{attribute 'reflection'}
FUNCTION_BLOCK FBEvent
VAR_INPUT
END_VAR
VAR_OUTPUT
END_VAR
VAR
  runner: REFERENCE TO EventRunner;
  {attribute 'instance-path'}
  {attribute 'noinit'}
  path: STRING(255);
  id: INT;
  _message: STRING(255);
END_VAR

METHOD add_message
VAR_INPUT
  level: EventLevel;
END_VAR
runner.add_message(id:=id, level:=level);
END_METHOD

METHOD alarm_raised : BOOL
VAR_INPUT
END_VAR
alarm_raised := runner.raised_history_count(id) > 0;
END_METHOD

METHOD clear_alarm
VAR_INPUT
END_VAR
runner.clear_alarm(id:=id);
END_METHOD

METHOD error_alarm
VAR_INPUT
END_VAR
raise_alarm(level:=EventLevel.ERROR);
END_METHOD

METHOD error_message
VAR_INPUT
END_VAR
add_message(level:=EventLevel.ERROR);
END_METHOD

METHOD FB_init : BOOL
VAR_INPUT
	bInitRetains : BOOL; // if TRUE, the retain variables are initialized (warm start / cold start)
	bInCopyCode : BOOL;  // if TRUE, the instance afterwards gets moved into the copy code (online change)
  runner: REFERENCE TO EventRunner;
END_VAR
IF __ISVALIDREF(runner) THEN
  runner.add_event(THIS^);
  THIS^.runner REF= runner;
END_IF
END_METHOD

METHOD info_alarm
VAR_INPUT
END_VAR
raise_alarm(level:=EventLevel.INFO);
END_METHOD

METHOD info_message
VAR_INPUT
END_VAR
add_message(level:=EventLevel.INFO);
END_METHOD

PROPERTY instance_path : STRING(255)
GET
instance_path := path;
END_GET
END_PROPERTY

PROPERTY message : STRING(255)
GET
message := _message;
END_GET
SET
_message := message;
END_SET
END_PROPERTY

METHOD raise_alarm
VAR_INPUT
  level: EventLevel;
END_VAR
runner.raise_alarm(id:=id, level:=level);
END_METHOD

METHOD INTERNAL set_id
VAR_INPUT
  id: INT;
END_VAR
THIS^.id := id;
END_METHOD

METHOD warning_alarm
VAR_INPUT
END_VAR
raise_alarm(level:=EventLevel.WARNING);
END_METHOD

METHOD warning_message
VAR_INPUT
END_VAR
add_message(level:=EventLevel.WARNING);
END_METHOD

END_FUNCTION_BLOCK

(* stored: Version 1.1.0.1, ProductVersion 3.1.4022.18
   POU FBEvent: Id {03cc76af-17ce-40eb-bb2a-7913c5ab3a91}, SpecialFunc None
   Method add_message: Id {5cbfa2c1-1c09-4567-9983-e434249344bc}
   Method alarm_raised: Id {d5a53cec-25bf-456d-9d29-f598e0a02060}
   Method clear_alarm: Id {7cc823d2-a8dd-44ff-903e-fdbcff90c798}
   Method error_alarm: Id {55e8d959-842f-4996-ac2c-8dd7cddc5c5b}
   Method error_message: Id {ca38d702-e59f-46d2-9511-1415bc78b78f}
   Method FB_init: Id {7731af07-9e97-4141-9829-41a64228a976}
   Method info_alarm: Id {ebd43a98-e667-4595-89c9-a229f5f0f0d6}
   Method info_message: Id {c0f9f1db-48a1-4979-bf36-bb8af0c33ed2}
   Property instance_path: Id {8a5a1c1c-ff06-4418-9b66-52ecf8d7f269}
   Get Get: Id {502f1fc3-998f-4e3e-ac0b-443913534009}
   Property message: Id {95b2f84d-eb7a-4759-a78c-209d6dcdc019}
   Get Get: Id {f93df829-d8fe-4832-a369-057f95411a5d}
   Set Set: Id {c521e5f0-7926-4ff9-9eb2-135493eb5d8f}
   Method raise_alarm: Id {b92c7d97-5a9f-4a9c-8999-52ff932d2446}
   Method set_id: Id {ca8e16af-abb6-4e45-b03a-925bd73ad678}
   Method warning_alarm: Id {f15a875c-59ec-43c3-b61d-c6f041445d2c}
   Method warning_message: Id {38bd0a24-bea0-4de5-869a-4f5133c97093} *)
